FUNCTION_BLOCK SomeTestPositions EXTENDS TcoDrivesBeckhoff.TcoSingleAxisPositionsRootContainer
VAR_INPUT
END_VAR
VAR_OUTPUT
END_VAR
VAR
	{attribute addProperty Name "<#Pick Position#>"}
	PickPosition:TcoDrivesBeckhoff.TcoSingleAxisMoveParam;
	{attribute addProperty Name "<#Place  Position#>"}
	PlacePosition:TcoDrivesBeckhoff.TcoSingleAxisMoveParam;
	{attribute addProperty Name "<#BlazkoPosition  Position#>"}
	BlazkoPosition:TcoDrivesBeckhoff.TcoSingleAxisMoveParam;
END_VAR

END_FUNCTION_BLOCK

(* stored: Version 1.1.0.1, ProductVersion 3.1.4024.12
   POU SomeTestPositions: Id {00d8b7c4-ef7f-03f9-2c3e-06b46cf10665}, SpecialFunc None *)
